PROGRAM MAIN
VAR
	Counter	:UDINT;
END_VAR

Counter:=Counter+1;

END_PROGRAM

(* stored: Version 1.1.0.1, ProductVersion 3.1.4024.12
   POU MAIN: Id {5f92e3a5-cf76-46ea-baeb-96201743b010}, SpecialFunc None *)
